{attribute 'qualified_only'}
{attribute 'strict'}
{attribute 'to_string'}
TYPE E_OPERATION_MODE :
(
	UNDEFINED,
	
	AUTO,

	MANUAL,
	
	MUST_BE_LAST	// ALWAYS KEEP THIS LAST!!!
);
END_TYPE

(* stored: Version 1.1.0.1, ProductVersion 3.1.4026.18
   DUT E_OPERATION_MODE: Id {fcb39d04-f77d-036d-0854-e470fda5f123} *)
